TYPE st_Router_Events :
STRUCT
	b_MBCommWarning		:	BOOL;
	b_NoSimWarning		:	BOOL;
	b_NoNetworkWarning	: 	BOOL;
	b_noGPSFixWarning	:	BOOL;
	b_SMSNotSendError	:	BOOL; 
	b_NoSMSNumberAvailable	:	BOOL;
	b_TimeUpdateFailed 	: BOOL;
END_STRUCT
END_TYPE

(* stored: Version 1.1.0.1, ProductVersion 3.1.4026.18
   DUT st_Router_Events: Id {cd092dc8-29f2-4e3d-a6b8-43e406070d5a} *)
